FUNCTION_BLOCK PAModule EXTENDS PAClassPhysicalBase
VAR_INPUT
END_VAR
VAR_OUTPUT
END_VAR
VAR
END_VAR

END_FUNCTION_BLOCK

(* stored: Version 1.1.0.1, ProductVersion 3.1.4020.12
   POU PAModule: Id {2c897f2d-db84-43c4-bcce-3e608c724a80}, SpecialFunc None *)
